(* IEC 61131-3 sources: CodesysTest/export/SX_1195.dev/Plc Logic/Application/PRJ Specific/Motion/Motors/Applied Motion/Applied Motion TSM34IP-3DG/Applied Motion TSM34IP-3DG Data Handlers/FB_StepServoCommands.pou/StopCrash.prop, 1 file *)

(* ---- Set.pm.st ---- *)
(*#-#-#-#-#-#-#-#-#-#---Declaration---#-#-#-#-#-#-#-#-#-#-#-#-#*)

VAR
END_VAR
(*#-#-#-#-#-#-#-#-#-#---Implementation---#-#-#-#-#-#-#-#-#-#-#-#-#*)

IF commandSuccessful THEN
	IF _previousCommandWord.14 <> 0 THEN
		_previousCommandWord := 0;
	ELSE
		commandSuccessful := FALSE;
		_stopAndKillCrash := StopCrash;
	END_IF
END_IF
